(* LS Electric XG5000 project: Study6_user_defined_functions *)
(* PLC LSPLC *)
(* module base 0 slot 0: 입력 모듈:XGI-D22A/B (DC 24V 입력, 16점 (전류소스 싱크공용/ 전류소스 입력)) *)
(* module base 0 slot 1: 출력 모듈:XGQ-RY2A/B (릴레이 출력, 16점 (2A용, Varistor 없음/Varistor 부착)) *)

FUNCTION ADDSUB : INT
VAR_INPUT
    Input1 : INT;
    Input2 : INT;
    Input3 : INT;
END_VAR
VAR
    add1 : INT;
END_VAR

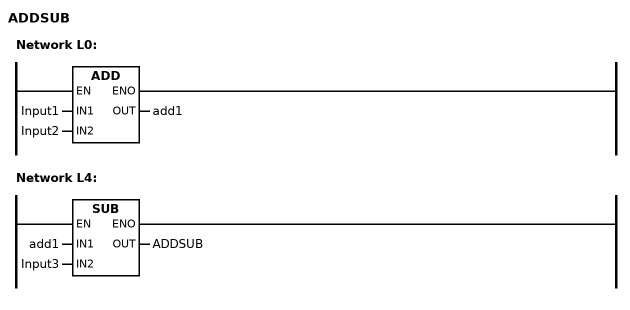
(* Rung L0 *)
add1 := Input1 + Input2;
(* Rung L4 *)
ADDSUB := add1 - Input3;
END_FUNCTION

FUNCTION ADDSUBDIV : INT
(* 사용자 정의 펑션 더하고 빼고 나누고 *)
VAR_INPUT
    input1 : INT;
    input2 : INT;
    input3 : INT;
    input4 : INT;
END_VAR
VAR_OUTPUT
    output1 : INT;
END_VAR
VAR
    output2 : INT;
END_VAR

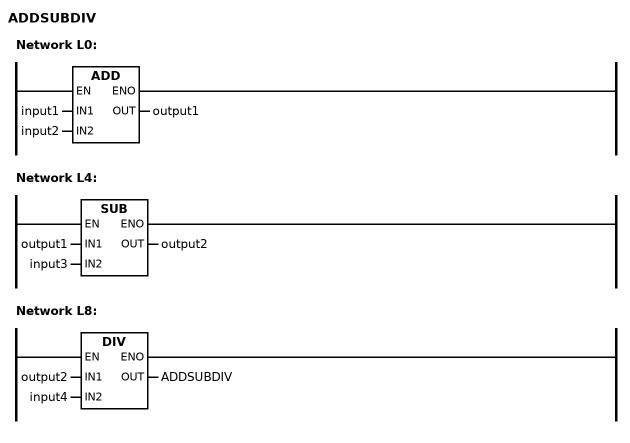
(* Rung L0 *)
output1 := input1 + input2;
(* Rung L4 *)
output2 := output1 - input3;
(* Rung L8 *)
ADDSUBDIV := output2 / input4;
END_FUNCTION

FUNCTION PITA : REAL
(* 피타고라스 함수 *)
VAR_INPUT
    A : REAL;
    B : REAL;
END_VAR
VAR
    addresult : REAL;
    As : REAL;
    Bs : REAL;
END_VAR

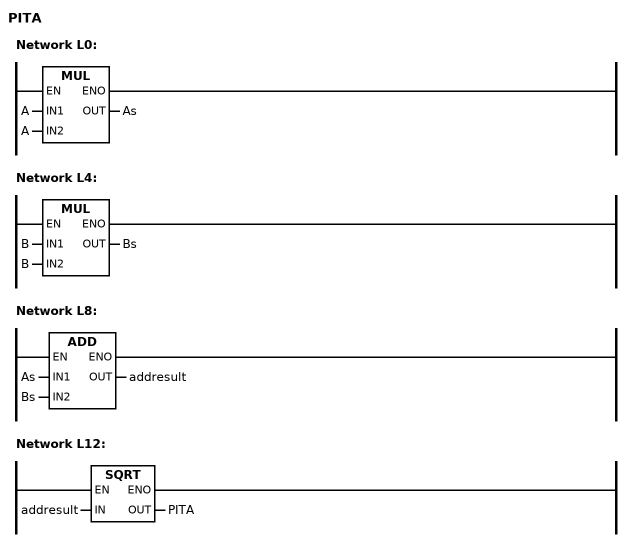
(* Rung L0 *)
As := A * A;
(* Rung L4 *)
Bs := B * B;
(* Rung L8 *)
addresult := As + Bs;
(* Rung L12 *)
PITA := SQRT(addresult);
END_FUNCTION

FUNCTION_BLOCK 사칙연산
VAR_INPUT
    A : INT;
    B : INT;
END_VAR
VAR_OUTPUT
    Add : INT;
    Sub : INT;
    Mul : INT;
    Div : INT;
END_VAR
VAR
    CV : INT;
    리셋 : BOOL;
    업카운터1 : CTU_INT;
    점멸횟수 : INT;
END_VAR

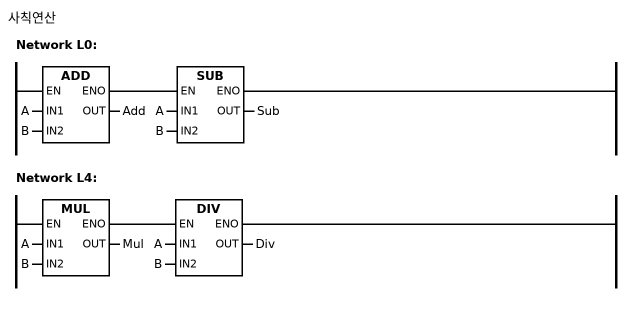
(* Rung L0 *)
Add := A + B;
Sub := A - B;
(* Rung L4 *)
Mul := A * B;
Div := A / B;
END_FUNCTION_BLOCK

FUNCTION_BLOCK 만능점멸기
(* 알아서 깜빡여주세요 *)
VAR_INPUT
    시작 : BOOL;
    시간간격 : TIME;
    점멸횟수 : INT;
END_VAR
VAR_OUTPUT
    출력 : BOOL;
END_VAR
VAR
    CV : INT;
    OUT : BOOL;
    Q : BOOL;
    리셋 : BOOL;
    업카운터1 : CTU_INT;
    오프타이머1 : TOF;
    온타이머1 : TON;
    온타이머2 : TON;
END_VAR
VAR
    _e1 : R_TRIG;
END_VAR

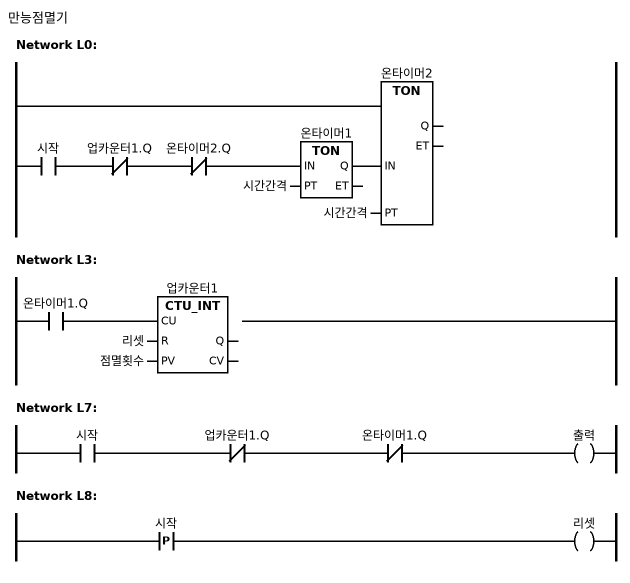
(* Rung L0 *)
온타이머1(IN := 시작 AND NOT 업카운터1.Q AND NOT 온타이머2.Q, PT := 시간간격);
온타이머2(IN := 온타이머1.Q, PT := 시간간격);
(* Rung L3 *)
업카운터1(CU := 온타이머1.Q, R := 리셋, PV := 점멸횟수);
(* Rung L7 *)
출력 := 시작 AND NOT 업카운터1.Q AND NOT 온타이머1.Q;
(* Rung L8 *)
_e1(CLK := 시작);
리셋 := _e1.Q;
END_FUNCTION_BLOCK

FUNCTION_BLOCK 오초깜빡이
VAR_INPUT
    FL : BOOL;
    NFL : BOOL;
    OFF : BOOL;
END_VAR
VAR_OUTPUT
    출력1 : BOOL;
    출력2 : BOOL;
END_VAR
VAR
    FL자가유지 : BOOL;
    NFL자가유지 : BOOL;
    타이머1 : TP;
    타이머2 : TP;
END_VAR

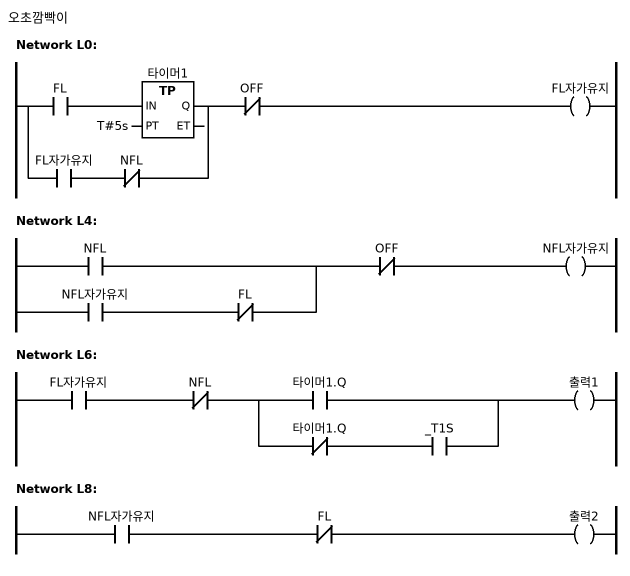
(* Rung L0 *)
타이머1(IN := FL, PT := T#5s);
FL자가유지 := (타이머1.Q OR (FL자가유지 AND NOT NFL)) AND NOT OFF;
(* Rung L4 *)
NFL자가유지 := (NFL OR (NFL자가유지 AND NOT FL)) AND NOT OFF;
(* Rung L6 *)
출력1 := FL자가유지 AND NOT NFL AND (타이머1.Q OR (NOT 타이머1.Q AND _T1S));
(* Rung L8 *)
출력2 := NFL자가유지 AND NOT FL;
END_FUNCTION_BLOCK

PROGRAM NewProgram (* task: 스캔 프로그램 *)
VAR
    FL : BOOL;
    FL자가유지 : BOOL;
    NFL : BOOL;
    NFL자가유지 : BOOL;
    OFF : BOOL;
    Output : INT;
    Output2 : INT;
    OutputPita : REAL;
    램프0 AT %QX0.1.0 : BOOL;
    램프1 AT %QX0.1.1 : BOOL;
    램프2 AT %QX0.1.2 : BOOL;
    리셋 : BOOL;
    사칙연산 : 사칙연산;
    시간간격 : TIME;
    시작 : BOOL;
    업카운터1 : CTU_INT;
    업타이머1 : TON;
    업타이머2 : TON;
    오초깜빡이 : 오초깜빡이;
    오프타이머1 : TOF;
    온오프 : BOOL;
    온타이머1 : TON;
    온타이머2 : TON;
    온타이머3 : TON;
    온타이머4 : TON;
    일초점등 : BOOL;
    일초점등스위치 : BOOL;
    입력1 : BOOL;
    입력2 : BOOL;
    점멸기 : 만능점멸기;
    점멸횟수 : INT;
    출력 : BOOL;
    출력1 : BOOL;
    출력2 : BOOL;
    타이머1 : TP;
    타이머2 : TP;
END_VAR

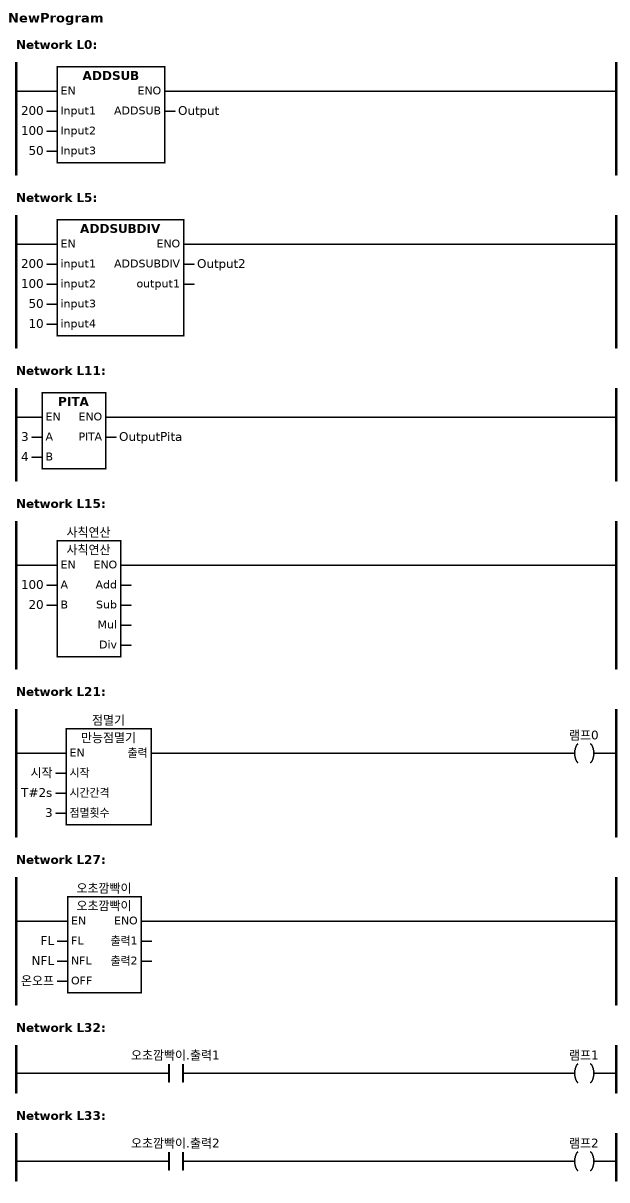
(* Rung L0 *)
Output := ADDSUB(Input1 := 200, Input2 := 100, Input3 := 50);
(* Rung L5 *)
Output2 := ADDSUBDIV(input1 := 200, input2 := 100, input3 := 50, input4 := 10);
(* Rung L11 *)
OutputPita := PITA(A := 3, B := 4);
(* Rung L15 *)
사칙연산(A := 100, B := 20);
(* Rung L21 *)
점멸기(시작 := 시작, 시간간격 := T#2s, 점멸횟수 := 3);
램프0 := 점멸기.출력;
(* Rung L27 *)
오초깜빡이(FL := FL, NFL := NFL, OFF := 온오프);
(* Rung L32 *)
램프1 := 오초깜빡이.출력1;
(* Rung L33 *)
램프2 := 오초깜빡이.출력2;
END_PROGRAM